PROGRAM MAIN
VAR
	bEingang:BOOL;
	sFirmaName:string;
	aArraya:ARRAY[1..80]OF BYTE;
END_VAR

END_PROGRAM

(* stored: Version 1.1.0.1, ProductVersion 3.1.4024.0
   POU MAIN: Id {62977ecd-ac31-43d2-8bc8-b9b1c617a583}, SpecialFunc None *)
